(*
	Allows direct reading of strings of arrays, inside a structure/function block/program, in a single read from C#
*)
TYPE ST_StringForArray :
STRUCT
	(* String for array *)
	str	: STRING;
END_STRUCT
END_TYPE

(* stored: Version 1.1.0.1
   DUT ST_StringForArray: Id {85d13bd0-d57c-4e92-b932-3870fbfcbe85} *)
